INTERFACE IPlugin

METHOD Run : BOOL
VAR_INPUT
END_VAR
END_METHOD

END_INTERFACE

(* stored: Version 1.1.0.1
   Itf IPlugin: Id {a90139af-c645-4465-a767-35d4a3a446d8}
   Method Run: Id {b378704d-347d-4262-8430-0027cb10569d} *)
